ABB RAPID module: 004609C8

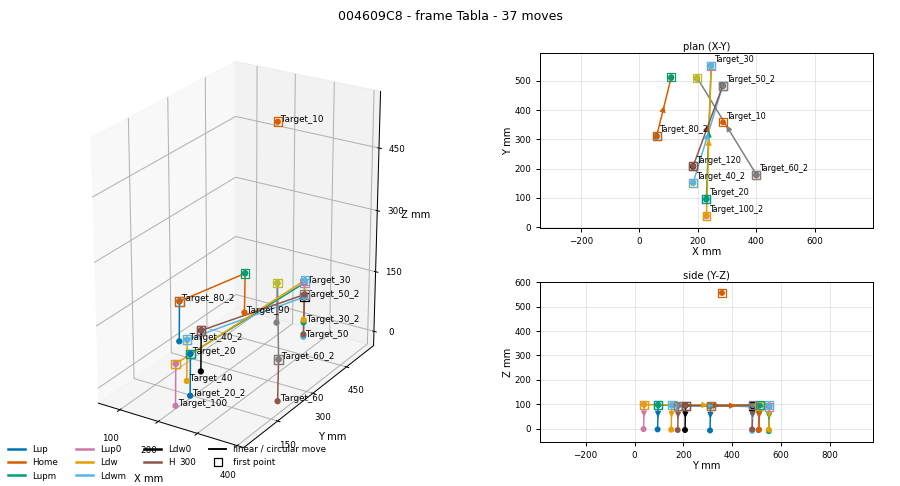
[picture p0: tool path of 004609C8 in frame Tabla, 37 of 37 moves have a stored position in this frame; points joined in program order, loops and branches not executed]
MODULE Module1
    CONST robtarget Target_20:=[[229.12374666,96.731764507,97.263749646],[0.005884839,0.38264087,-0.923826969,0.00975011],[-1,0,-2,0],[9E+09,9E+09,9E+09,9E+09,9E+09,9E+09]];
    CONST robtarget Target_20_2:=[[228.782590129,94.479925502,-2.710311156],[0.005884839,0.38264087,-0.923826969,0.00975011],[-1,0,-2,0],[9E+09,9E+09,9E+09,9E+09,9E+09,9E+09]];
    CONST robtarget Target_10:=[[286.192182184,358.139537963,556.107701921],[0.171957146,-0.001936356,0.985040077,-0.011092229],[0,0,0,0],[9E+09,9E+09,9E+09,9E+09,9E+09,9E+09]];
    CONST robtarget Target_30:=[[245.510885963,551.88763337,89.95657104],[0.005884839,0.38264087,-0.923826969,0.00975011],[0,1,-2,0],[9E+09,9E+09,9E+09,9E+09,9E+09,9E+09]];
    CONST robtarget Target_30_2:=[[245.169729432,549.635794365,-10.017489763],[0.005884839,0.38264087,-0.923826969,0.00975011],[0,1,-2,0],[9E+09,9E+09,9E+09,9E+09,9E+09,9E+09]];
    CONST robtarget Target_40_2:=[[184.040008961,152.340124362,96.165060034],[0.005884839,0.38264087,-0.923826969,0.00975011],[-1,1,-2,0],[9E+09,9E+09,9E+09,9E+09,9E+09,9E+09]];
    CONST robtarget Target_40:=[[183.69885248,150.088285465,-3.809000771],[0.005884839,0.38264087,-0.923826969,0.00975011],[-1,1,-2,0],[9E+09,9E+09,9E+09,9E+09,9E+09,9E+09]];
    CONST robtarget Target_50_2:=[[285.049655836,483.705888558,91.357388428],[0.007029214,0.492374909,-0.870308711,0.008960253],[0,0,-2,0],[9E+09,9E+09,9E+09,9E+09,9E+09,9E+09]];
    CONST robtarget Target_50:=[[284.708499352,481.454049588,-8.616672375],[0.007029214,0.492374909,-0.870308711,0.008960253],[0,1,-2,0],[9E+09,9E+09,9E+09,9E+09,9E+09,9E+09]];
    CONST robtarget Target_60_2:=[[400.096751677,179.051746899,94.826118299],[0.005884839,0.38264087,-0.923826969,0.00975011],[-1,0,-1,0],[9E+09,9E+09,9E+09,9E+09,9E+09,9E+09]];
    CONST robtarget Target_60:=[[399.755595146,176.799907894,-5.147942503],[0.005884839,0.38264087,-0.923826969,0.00975011],[-1,0,-2,0],[9E+09,9E+09,9E+09,9E+09,9E+09,9E+09]];
    CONST robtarget Target_70_2:=[[197.720398886,509.773560591,94.069019261],[0.004287134,0.233411549,-0.972311346,0.010550662],[0,-1,0,1],[9E+09,9E+09,9E+09,9E+09,9E+09,9E+09]];
    CONST robtarget Target_70:=[[197.37924231,507.521721572,-5.905041541],[0.004287134,0.233411549,-0.972311346,0.010550662],[0,-1,0,1],[9E+09,9E+09,9E+09,9E+09,9E+09,9E+09]];
    CONST robtarget Target_80_2:=[[59.200735476,311.399373985,93.008380327],[0.011259958,0.99993515,-0.000019207,-0.001705677],[-1,1,-1,1],[9E+09,9E+09,9E+09,9E+09,9E+09,9E+09]];
    CONST robtarget Target_80:=[[58.859578945,309.14753498,-6.965680475],[0.011259958,0.99993515,-0.000019207,-0.001705677],[-1,1,-1,1],[9E+09,9E+09,9E+09,9E+09,9E+09,9E+09]];
    CONST robtarget Target_90_2:=[[108.933738622,512.046855311,96.321314041],[0.009168088,0.707047344,-0.707074507,0.006755897],[0,-2,0,1],[9E+09,9E+09,9E+09,9E+09,9E+09,9E+09]];
    CONST robtarget Target_90:=[[108.592582168,509.795016351,-3.652746763],[0.009168088,0.707047344,-0.707074507,0.006755897],[0,-2,0,1],[9E+09,9E+09,9E+09,9E+09,9E+09,9E+09]];
    CONST robtarget Target_100_2:=[[229.439744782,39.245320884,98.557509349],[0.005884839,0.38264087,-0.923826969,0.00975011],[-1,0,-2,0],[9E+09,9E+09,9E+09,9E+09,9E+09,9E+09]];
    CONST robtarget Target_100:=[[229.098588301,36.993481987,-1.416551456],[0.005884839,0.38264087,-0.923826969,0.00975011],[-1,0,-2,0],[9E+09,9E+09,9E+09,9E+09,9E+09,9E+09]];
    CONST robtarget Target_110_2:=[[245.330356475,552.326681957,95.94885461],[0.005884839,0.38264087,-0.923826969,0.00975011],[0,1,-2,0],[9E+09,9E+09,9E+09,9E+09,9E+09,9E+09]];
    CONST robtarget Target_110:=[[244.989199994,550.07484306,-4.025206195],[0.005884839,0.38264087,-0.923826969,0.00975011],[0,1,-2,0],[9E+09,9E+09,9E+09,9E+09,9E+09,9E+09]];
    CONST robtarget Target_120_2:=[[184.040008951,208.925772071,94.89051174],[0.005884839,0.38264087,-0.923826969,0.00975011],[-1,0,2,0],[9E+09,9E+09,9E+09,9E+09,9E+09,9E+09]];
    CONST robtarget Target_120:=[[183.69885247,206.673933174,-5.083549065],[0.005884839,0.38264087,-0.923826969,0.00975011],[-1,1,2,0],[9E+09,9E+09,9E+09,9E+09,9E+09,9E+09]];
    CONST robtarget Target_130_2:=[[285.070125228,483.840998898,97.355832076],[0.007029214,0.492374909,-0.870308711,0.008960253],[0,0,-2,0],[9E+09,9E+09,9E+09,9E+09,9E+09,9E+09]];
    CONST robtarget Target_130:=[[284.728968744,481.589159928,-2.618228727],[0.007029214,0.492374909,-0.870308711,0.008960253],[0,1,-2,0],[9E+09,9E+09,9E+09,9E+09,9E+09,9E+09]];

    PROC main()
        Home;
        Lup;
        Lupm;
        Lup0;
        Ldw;
        Ldwm;
        Ldw0;
        H;
        Hm;
        H0;
        Lup3;
        Lup3m;
        Lup30;
        Ldw3;
        Ldw3m;
        Ldw30;
        Home;
    ENDPROC

    PROC Lup()
        MoveL Target_20,v200,z30,succión\WObj:=Tabla;
        MoveL Target_20_2,v200,z30,succión\WObj:=Tabla;
    ENDPROC
    PROC Home()
        MoveL Target_10,v200,z30,succión\WObj:=Tabla;
    ENDPROC
    PROC Lupm()
        MoveL Target_20,v200,z30,succión\WObj:=Tabla;
        MoveL Target_30,v200,z30,succión\WObj:=Tabla;
        MoveL Target_30_2,v200,z30,succión\WObj:=Tabla;
    ENDPROC
    PROC Lup0()
        MoveL Target_30,v200,z30,succión\WObj:=Tabla;
    ENDPROC
    PROC Ldw()
        MoveL Target_40_2,v200,z30,succión\WObj:=Tabla;
        MoveL Target_40,v200,z30,succión\WObj:=Tabla;
    ENDPROC
    PROC Ldwm()
        MoveL Target_40_2,v200,z30,succión\WObj:=Tabla;
        MoveL Target_50_2,v200,z30,succión\WObj:=Tabla;
        MoveL Target_50,v200,z30,succión\WObj:=Tabla;
    ENDPROC
    PROC Ldw0()
        MoveL Target_50_2,v200,z30,succión\WObj:=Tabla;
    ENDPROC
    PROC H()
        MoveL Target_60_2,v200,z30,succión\WObj:=Tabla;
        MoveL Target_60,v200,z30,succión\WObj:=Tabla;
    ENDPROC
    PROC Hm()
        MoveL Target_60_2,v200,z30,succión\WObj:=Tabla;
        MoveL Target_70_2,v200,z30,succión\WObj:=Tabla;
        MoveL Target_70,v200,z30,succión\WObj:=Tabla;
    ENDPROC
    PROC H0()
        MoveL Target_70_2,v200,z30,succión\WObj:=Tabla;
    ENDPROC
    PROC L()
        MoveL Target_80_2,v200,z30,succión\WObj:=Tabla;
        MoveL Target_80,v200,z30,succión\WObj:=Tabla;
    ENDPROC
    PROC Lm()
        MoveL Target_80_2,v200,z30,succión\WObj:=Tabla;
        MoveL Target_90_2,v200,z30,succión\WObj:=Tabla;
        MoveL Target_90,v200,z30,succión\WObj:=Tabla;
    ENDPROC
    PROC L0()
        MoveL Target_90_2,v200,z30,succión\WObj:=Tabla;
    ENDPROC
    PROC Lup3()
        MoveL Target_100_2,v200,z30,succión\WObj:=Tabla;
        MoveL Target_100,v200,z30,succión\WObj:=Tabla;
    ENDPROC
    PROC Lup3m()
        MoveL Target_100_2,v200,z30,succión\WObj:=Tabla;
        MoveL Target_110_2,v200,z30,succión\WObj:=Tabla;
        MoveL Target_110,v200,z30,succión\WObj:=Tabla;
    ENDPROC
    PROC Lup30()
        MoveL Target_110_2,v200,z30,succión\WObj:=Tabla;
    ENDPROC
    PROC Ldw3()
        MoveL Target_120_2,v200,z30,succión\WObj:=Tabla;
        MoveL Target_120,v200,z30,succión\WObj:=Tabla;
    ENDPROC
    PROC Ldw3m()
        MoveL Target_120_2,v200,z30,succión\WObj:=Tabla;
        MoveL Target_130_2,v200,z30,succión\WObj:=Tabla;
        MoveL Target_130,v200,z30,succión\WObj:=Tabla;
    ENDPROC
    PROC Ldw30()
        MoveL Target_130_2,v200,z30,succión\WObj:=Tabla;
    ENDPROC
ENDMODULE
